(* CODESYS project LD2_PROGRAMM.xml

Project tree, tasks and I/O mapping:
  program LD2_PROGRAMM [?]
*)

// LD2_PROGRAMM
PROGRAM LD2_PROGRAMM
VAR
	xStart : BOOL;
	xStop_NC : BOOL;
	xPump : BOOL;
	xLamp : BOOL;
	
	timer : TON;
END_VAR

(* body of a kind this reader does not render *)

END_PROGRAM
